FUNCTION "fcStdReportBatchStart" : Bool   // FC510, SCL
TITLE = Standard batch report start
{ S7_Optimized_Access := 'FALSE' }
AUTHOR : Boris
VERSION : 2.0
// 10/01/08 BC - Function needs to be called at batch start
//  Constant, used in all standard report FB and FC
   VAR_INPUT
      iInLineNo : Int;   // Line number
      iInMixerNo : Int;   // Mixer number
      sInFormulaName : String[254];   // Recipe name
      sInFormulaDescription : String[254];   // Recipe Description
      iInFormulaID : Int;   // Recipe ID
      iInBatchNumber : Int;   // Batch number
      sInTimeStart : String[254];   // Start timestamp
      rInMixerTempStart : Real;   // Mixer temperature AT batch start
   END_VAR
   VAR_IN_OUT
      MixerReportOperation : "udtStdReportOperV2";   // Current report operation with header and status
   END_VAR
   VAR_TEMP
      iTemp : Int;
      bResult : Bool;
   END_VAR
   VAR CONSTANT
      ciMaxQueue : Int := 200;   // Elements in the queue
      ciMaxUID : Int := 30000;
      ciReportDisable : Int;   // Not ready
      ciReportReady : Int := 10;   // Ready to save to database
      ciReportSavingToDataBase : Int := 20;   // Saving in progress
      ciReportFailed : Int := 30;   // Saving failed
      ciReportSaved : Int := 40;   // Saved
   END_VAR
BEGIN

       // Write batch header (with UID) to the mixer report operation header
       #MixerReportOperation.iBatchUID := "fcStdReportNewBatchUID"(); // Generate new global batch uid
       #MixerReportOperation.Header.iLineNo := #iInLineNo;
       #MixerReportOperation.Header.iMixerNo := #iInMixerNo;
       #MixerReportOperation.Header.iStatus := 220; // Set batch in progress status
       #iTemp := BLKMOV (DSTBLK => #MixerReportOperation.Header.sName, SRCBLK := #sInFormulaName);
       #iTemp := BLKMOV (DSTBLK => #MixerReportOperation.Header.sDescription, SRCBLK := #sInFormulaDescription);    
       #MixerReportOperation.Header.iRecipeID := #iInFormulaID;
       #MixerReportOperation.Header.iBatchNumber := #iInBatchNumber;
       #iTemp := BLKMOV (DSTBLK => #MixerReportOperation.Header.sTimeStart, SRCBLK := #sInTimeStart);        
       #MixerReportOperation.Header.rMixerTemp := #rInMixerTempStart;

       // Clear command structure
       #MixerReportOperation.Command.iStep := 0;
       #MixerReportOperation.Command.iStatus := 0;
       #MixerReportOperation.Command.sName := "sEmpty";
       #MixerReportOperation.Command.iCode := 0;
       #MixerReportOperation.Command.iIngredientType := 0;
       #MixerReportOperation.Command.sTimeStart := "sEmpty";
       #MixerReportOperation.Command.sTimeFinish := "sEmpty";
       #MixerReportOperation.Command.rSetpoint := 0.0;
       #MixerReportOperation.Command.rActual := 0.0;
       #MixerReportOperation.Command.rTemperature := 0.0;

       // Clear footer structure
       #MixerReportOperation.Footer.iStatus := 0;
       #MixerReportOperation.Footer.rMixerTemp := 0.0;
       #MixerReportOperation.Footer.sTimeFinish := "sEmpty";

       // Set reporting status to report ready
       #MixerReportOperation.iReportingStatus := #ciReportReady;

       // Generate new global index to write    
       #iTemp := "fcStdReportGetWriteIndex"();            
       // Check queue index already used, return false from function to indicate error
       IF ("dbStdReportQueueV2".Operations["dbStdReportQueueV2".iIndexWrite].iReportingStatus = #ciReportSaved) OR ("dbStdReportQueueV2".Operations["dbStdReportQueueV2".iIndexWrite].iReportingStatus = #ciReportDisable) THEN
           #bResult := true;
       ELSE
           #bResult := false;
       END_IF;

       // Write batch header to the queue
       #iTemp := BLKMOV (DSTBLK => "dbStdReportQueueV2".Operations["dbStdReportQueueV2".iIndexWrite], SRCBLK := #MixerReportOperation);

       // Return false if overwriting previous report in the queue
       #fcStdReportBatchStart := #bResult;                                
       ENO := true;
END_FUNCTION

FUNCTION "fcStdReportBatchComplete" : Bool   // FC511, SCL
TITLE = Standard batch report complete
{ S7_Optimized_Access := 'FALSE' }
AUTHOR : Boris
VERSION : 2.0
// 10/01/08 BC - Function needs to be called at batch complete
//  Constant, used in all standard report FB and FC
   VAR_INPUT
      iInLineNo : Int;   // Line number
      iInMixerNo : Int;   // Mixer number
      rInMixerTempFinish : Real;   // Mixer temperature
      sInTimeFinish : String[254];   // Complete timestamp
      iInBatchStatus : Int;   // Batch status (if not yet set)
   END_VAR
   VAR_IN_OUT
      MixerReportOperation : "udtStdReportOperV2";   // Current report operation with header and status
   END_VAR
   VAR_TEMP
      iTemp : Int;
      bResult : Bool;
   END_VAR
   VAR CONSTANT
      ciMaxQueue : Int := 200;   // Elements in the queue
      ciMaxUID : Int := 30000;
      ciReportDisable : Int;   // Not ready
      ciReportReady : Int := 10;   // Ready to save to database
      ciReportSavingToDataBase : Int := 20;   // Saving in progress
      ciReportFailed : Int := 30;   // Saving failed
      ciReportSaved : Int := 40;   // Saved
   END_VAR
BEGIN

       // Check batchUID, generate new if needed
       IF (#MixerReportOperation.iBatchUID = 0) THEN
           // Something went wrong - batch completed, but BatchUID is not set
           // Most likely it will be empty batch with only footer
           #MixerReportOperation.iBatchUID := "fcStdReportNewBatchUID"(); // Generate new global batch uid
           #MixerReportOperation.Header.iStatus := 220; // Set header to InProgress
       END_IF;

       // Clear command structure
       #MixerReportOperation.Command.iStep := 0;
       #MixerReportOperation.Command.iStatus := 0;
       #MixerReportOperation.Command.sName := "sEmpty";
       #MixerReportOperation.Command.iCode := 0;
       #MixerReportOperation.Command.iIngredientType := 0;
       #MixerReportOperation.Command.sTimeStart := "sEmpty";
       #MixerReportOperation.Command.sTimeFinish := "sEmpty";
       #MixerReportOperation.Command.rSetpoint := 0.0;
       #MixerReportOperation.Command.rActual := 0.0;
       #MixerReportOperation.Command.rTemperature := 0.0;

       // Write foter structure to the mixer operation report strucuture
       // If status not set yet - set it. Keep old status if it was previously set
       IF (#MixerReportOperation.Footer.iStatus = 0) THEN
           #MixerReportOperation.Footer.iStatus := #iInBatchStatus;
       END_IF;
       #MixerReportOperation.Footer.rMixerTemp := #rInMixerTempFinish;
       #iTemp := BLKMOV (DSTBLK => #MixerReportOperation.Footer.sTimeFinish, SRCBLK := #sInTimeFinish);                             
       #MixerReportOperation.Header.iLineNo := #iInLineNo;
       #MixerReportOperation.Header.iMixerNo := #iInMixerNo;

       // Set reporting status to report ready
       #MixerReportOperation.iReportingStatus := #ciReportReady;

       // Generate new global index to write    
       #iTemp := "fcStdReportGetWriteIndex"();  
       // Check queue index already used, return false from function to indicate error
       IF ("dbStdReportQueueV2".Operations["dbStdReportQueueV2".iIndexWrite].iReportingStatus = #ciReportSaved) OR ("dbStdReportQueueV2".Operations["dbStdReportQueueV2".iIndexWrite].iReportingStatus = #ciReportDisable) THEN
           #bResult := true;
       ELSE
           #bResult := false;
       END_IF;

       // Write batch header to the queue
       #iTemp := BLKMOV (DSTBLK => "dbStdReportQueueV2".Operations["dbStdReportQueueV2".iIndexWrite], SRCBLK := #MixerReportOperation);

       // Clear mixer operation report header strucutre
       #MixerReportOperation.iBatchUID := 0;
       #MixerReportOperation.Header.iLineNo := #iInLineNo;
       #MixerReportOperation.Header.iMixerNo := #iInMixerNo;
       #MixerReportOperation.Header.sName := "sEmpty";
       #MixerReportOperation.Header.sDescription := "sEmpty";
       #MixerReportOperation.Header.iRecipeID := 0;
       #MixerReportOperation.Header.iBatchNumber := 0;
       #MixerReportOperation.Header.iStatus := 0;
       #MixerReportOperation.Header.sTimeStart := "sEmpty";
       #MixerReportOperation.Header.rMixerTemp := 0.0;

       // Clear footer structure
       #MixerReportOperation.Footer.iStatus := 0;
       #MixerReportOperation.Footer.rMixerTemp := 0.0;
       #MixerReportOperation.Footer.sTimeFinish := "sEmpty";

       #MixerReportOperation.iReportingStatus := 0;

       // Return false if overwriting previous report in the queue
       #fcStdReportBatchComplete := #bResult;                                  
       ENO := true;
END_FUNCTION

FUNCTION "fcStdReportOper" : Bool   // FC512, SCL
TITLE = Standard batch report store operation
{ S7_Optimized_Access := 'FALSE' }
AUTHOR : Boris
VERSION : 2.0
// 10/01/08 BC - Function needs to be called at batch complete
//  Constant, used in all standard report FB and FC
   VAR_INPUT
      iInLineNo : Int;   // Line number
      iInMixerNo : Int;   // Mixer number
      iInStepNumber : Int;   // Command step number (0 if outside the recipe)
      iInCommandStatus : Int;   // Command delivery status
      sInCommandName : String[254];   // Command/Ingredient string name
      iInCommandCode : Int;   // Comand/Ingredient code
      iInCommandIngredientType : Int;   // Igredient type code
      sInCommandTimeStart : String[254];   // Delivery start time string
      sInCommandTimeFinish : String[254];   // Delivery comlete time string
      rInCommandSetpoint : Real;   // Delivery set point
      rInCommandActual : Real;   // Delivered actual
      rInCommandTemperature : Real;   // Ingredient temperature
   END_VAR
   VAR_IN_OUT
      MixerReportOperation : "udtStdReportOperV2";   // Current report operation with header and status
   END_VAR
   VAR_TEMP
      iTemp : Int;
      bResult : Bool;
   END_VAR
   VAR CONSTANT
      ciMaxQueue : Int := 200;   // Elements in the queue
      ciMaxUID : Int := 30000;
      ciReportDisable : Int;   // Not ready
      ciReportReady : Int := 10;   // Ready to save to database
      ciReportSavingToDataBase : Int := 20;   // Saving in progress
      ciReportFailed : Int := 30;   // Saving failed
      ciReportSaved : Int := 40;   // Saved
   END_VAR
BEGIN

       // Check batchUID, generate new if needed
       IF (#MixerReportOperation.iBatchUID = 0) THEN
           // Looks like we running test ingredient recipe
           #MixerReportOperation.Header.iStatus := 200; // Set header to TestRecipe
       END_IF;

       // Not normal situation - header status not set, assume test ingredient
       IF (#MixerReportOperation.Header.iStatus = 0) THEN
           #MixerReportOperation.Header.iStatus := 200; // Set header to TestRecipe
       END_IF;

       // Check if we running test recipe, idicated by header status
       IF (#MixerReportOperation.Header.iStatus = 200) THEN
           // Check if it's not intermediate weight        
           IF (#MixerReportOperation.Command.iStatus <> 1000) THEN    
               #iTemp := "fcStdReportNewBatchUID"(); // Generate new global batch uid
           END_IF;

           // Clear mixer operation report header structure
           #MixerReportOperation.Header.sName := "sEmpty";
           #MixerReportOperation.Header.sDescription := "sEmpty";
           #MixerReportOperation.Header.iRecipeID := 0;
           #MixerReportOperation.Header.iBatchNumber := 0;
           #MixerReportOperation.Header.sTimeStart := "sEmpty";
           #MixerReportOperation.Header.rMixerTemp := 0.0;

           // Clear footer structure        
           #MixerReportOperation.Footer.iStatus := 0;
           #MixerReportOperation.Footer.rMixerTemp := 0.0;
           #MixerReportOperation.Footer.sTimeFinish := "sEmpty";
       END_IF;

       // Set batch header 
       #MixerReportOperation.Header.iLineNo := #iInLineNo;
       #MixerReportOperation.Header.iMixerNo := #iInMixerNo;

       // Write command structure to the Mixer report operation structure
       #MixerReportOperation.Command.iStep := #iInStepNumber;
       #MixerReportOperation.Command.iStatus := #iInCommandStatus;
       #iTemp := BLKMOV (DSTBLK => #MixerReportOperation.Command.sName, SRCBLK := #sInCommandName);
       #MixerReportOperation.Command.iCode := #iInCommandCode;
       #MixerReportOperation.Command.iIngredientType := #iInCommandIngredientType;
       #iTemp := BLKMOV (DSTBLK => #MixerReportOperation.Command.sTimeStart, SRCBLK := #sInCommandTimeStart);
       #iTemp := BLKMOV (DSTBLK => #MixerReportOperation.Command.sTimeFinish, SRCBLK := #sInCommandTimeFinish);
       #MixerReportOperation.Command.rSetpoint := #rInCommandSetpoint;
       #MixerReportOperation.Command.rActual := #rInCommandActual;
       #MixerReportOperation.Command.rTemperature := #rInCommandTemperature;                                

       // Set reporting status to report ready
       #MixerReportOperation.iReportingStatus := #ciReportReady;

       // Generate new global index to write    
       #iTemp := "fcStdReportGetWriteIndex"();    
       // Check queue index already used, return false from function to indicate error
       IF ("dbStdReportQueueV2".Operations["dbStdReportQueueV2".iIndexWrite].iReportingStatus = #ciReportSaved) OR ("dbStdReportQueueV2".Operations["dbStdReportQueueV2".iIndexWrite].iReportingStatus = #ciReportDisable) THEN
           #bResult := true;
       ELSE
           #bResult := false;
       END_IF;

       // Write batch header to the queue
       #iTemp := BLKMOV (DSTBLK => "dbStdReportQueueV2".Operations["dbStdReportQueueV2".iIndexWrite], SRCBLK := #MixerReportOperation);

       // Return false if overwriting previous report in the queue
       #fcStdReportOper := #bResult;                 
       ENO := true;
END_FUNCTION

FUNCTION "fcStdReportBatchStatus" : Void   // FC513, SCL
TITLE = Standard batch report set batch status
{ S7_Optimized_Access := 'FALSE' }
AUTHOR : Boris
VERSION : 2.0
// Constant, used in all standard report FB and FC
   VAR_INPUT
      iInLineNo : Int;   // Line number
      iInMixerNo : Int;   // Mixer number
      iInBatchStatus : Int;   // Batch status to set
   END_VAR
   VAR_IN_OUT
      MixerReportOperation : "udtStdReportOperV2";   // Current report operation with header and status
   END_VAR
   VAR_TEMP
      iTemp : Int;
      bResult : Bool;
   END_VAR
   VAR CONSTANT
      ciMaxQueue : Int := 200;   // Elements in the queue
      ciMaxUID : Int := 30000;
      ciReportDisable : Int;   // Not ready
      ciReportReady : Int := 10;   // Ready to save to database
      ciReportSavingToDataBase : Int := 20;   // Saving in progress
      ciReportFailed : Int := 30;   // Saving failed
      ciReportSaved : Int := 40;   // Saved
   END_VAR
BEGIN

       // Write batch header
       #MixerReportOperation.Header.iLineNo := #iInLineNo;
       #MixerReportOperation.Header.iMixerNo := #iInMixerNo;

       // If status not set yet - set it. Keep old status if it was previously set
       IF (#MixerReportOperation.Footer.iStatus = 0) THEN
           #MixerReportOperation.Footer.iStatus := #iInBatchStatus;
       END_IF;

       ENO := true;
END_FUNCTION

FUNCTION "fcStdReportNewBatchUID" : Int   // FC514, SCL
TITLE = Standard batch report generates and return new batchUID
{ S7_Optimized_Access := 'FALSE' }
AUTHOR : Boris
VERSION : 2.0
// Constant, used in all standard report FB and FC
   VAR_TEMP
      i : Int;
   END_VAR
   VAR CONSTANT
      ciMaxQueue : Int := 200;   // Elements in the queue
      ciMaxUID : Int := 30000;
      ciReportDisable : Int;   // Not ready
      ciReportReady : Int := 10;   // Ready to save to database
      ciReportSavingToDataBase : Int := 20;   // Saving in progress
      ciReportFailed : Int := 30;   // Saving failed
      ciReportSaved : Int := 40;   // Saved
   END_VAR
BEGIN

       // Generate new global batch uid
       #i := "dbStdReportQueueV2".iGlobalBatchUID + 1;
       IF (#i > #ciMaxUID) THEN
          #i := 1;
       END_IF;  
       "dbStdReportQueueV2".iGlobalBatchUID := #i;

       #fcStdReportNewBatchUID := "dbStdReportQueueV2".iGlobalBatchUID;
       ENO := true;
END_FUNCTION

FUNCTION "fcStdReportGetWriteIndex" : Int   // FC515, SCL
TITLE = Standard batch report get queue write index
{ S7_Optimized_Access := 'FALSE' }
AUTHOR : Boris
VERSION : 2.0
// Constant, used in all standard report FB and FC
   VAR_TEMP
      i : Int;
   END_VAR
   VAR CONSTANT
      ciMaxQueue : Int := 200;   // Elements in the queue
      ciMaxUID : Int := 30000;
      ciReportDisable : Int;   // Not ready
      ciReportReady : Int := 10;   // Ready to save to database
      ciReportSavingToDataBase : Int := 20;   // Saving in progress
      ciReportFailed : Int := 30;   // Saving failed
      ciReportSaved : Int := 40;   // Saved
   END_VAR
BEGIN

       // Generate new global index to write    
       #i := "dbStdReportQueueV2".iIndexWrite + 1;      
       // Check queue index at the end of the queue
       IF (#i > #ciMaxQueue) THEN
           #i := 1;
       END_IF;               
       "dbStdReportQueueV2".iIndexWrite := #i;           

       #fcStdReportGetWriteIndex := "dbStdReportQueueV2".iIndexWrite;
       ENO := true;
END_FUNCTION

// folder: Resources/Process

FUNCTION_BLOCK "fbRetentiveTimer"   // FB385, LAD
TITLE = Retentive Timer Block
{ S7_Optimized_Access := 'TRUE' }
AUTHOR : DMC
FAMILY : LowLevel
VERSION : 0.1
// //  This is a retentive count-up timer.
// //  IN makes it count.  It does not reset when IN is off.
// //  RESET resets the time to 0.  
// //  bInPT is the time setpoint.
// //  bOutEnabled is true when the time has the setpoint
// //  bOutET is the elapsed time.
   VAR_INPUT
      IN : Bool;   // Counter Starts when this is true
      RESET : Bool;   // Counter Resets when this is true
      PT : Time;   // Time setpoint
   END_VAR
   VAR_OUTPUT
      Q : Bool;   // True when Elapsed time > Time Setpoint
      ET : Time;   // Elapsed Time
   END_VAR
   VAR
      "Timer" : IEC_TIMER;   // Timer
      tInternalTime : Time;   // Internal Time
      tTimer1ET : Time;   // Elapsed Time of Timer 1
      ET_DINT : DInt;   // Elapsed Time as a double integer
      bTON_Timer : Bool;
   END_VAR
   VAR_TEMP
      diTemp1 : DInt;   // Temp Double int
      diTemp2 : DInt;   // Temp Double int
      diTemp3 : DInt;   // Temp Double int
      tTemp : Time;
   END_VAR
   VAR CONSTANT
      ctMaxTime : Time := T#24D_20H_31M_23S_647MS;   // Max possible time
   END_VAR
BEGIN

REGION Network 1: Keep resetting internal time while not counting
   // IF (NOT IN) THEN
   //     tInternalTime := tInternalTime + Timer1.ET;
   // END_IF;
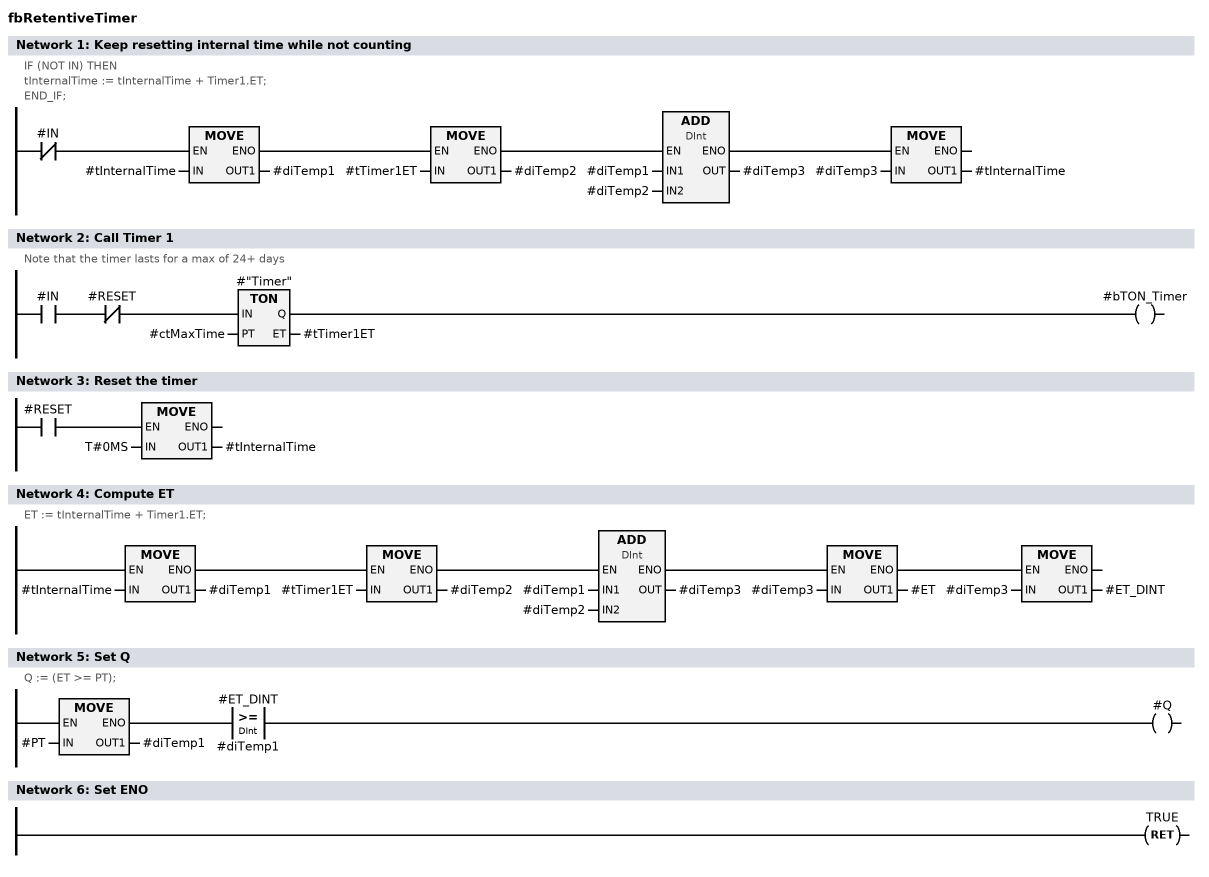
   RUNG wire#powerrail
      I_Contact( #IN )
      { S7_GenerateENO := "TRUE" } Move(in := #tInternalTime, out1 => #diTemp1)
      { S7_GenerateENO := "TRUE" } Move(in := #tTimer1ET, out1 => #diTemp2)
      { S7_Templates := "SrcType := DInt"; S7_GenerateENO := "TRUE" } Add(in1 := #diTemp1, in2 := #diTemp2, out => #diTemp3)
      { S7_GenerateENO := "TRUE" } Move(in := #diTemp3, out1 => #tInternalTime)
   END_RUNG
   // the same network as SCL:
   // ENO of a box is taken as its EN; it also drops when the box reports an error
   IF NOT #IN THEN
       #diTemp1 := #tInternalTime;
       #diTemp2 := #tTimer1ET;
       #diTemp3 := #diTemp1 + #diTemp2;
       #tInternalTime := #diTemp3;
   END_IF;
END_REGION

REGION Network 2: Call Timer 1
   // Note that the timer lasts for a max of 24+ days
   #"Timer".TON(IN := #IN AND NOT #RESET, PT := #ctMaxTime, ET => #tTimer1ET);
   #bTON_Timer := #"Timer".Q;
END_REGION

REGION Network 3: Reset the timer
   RUNG wire#powerrail
      Contact( #RESET )
      { S7_GenerateENO := "TRUE" } Move(in := T#0MS, out1 => #tInternalTime)
   END_RUNG
   // the same network as SCL:
   IF #RESET THEN #tInternalTime := T#0MS; END_IF;
END_REGION

REGION Network 4: Compute ET
   // ET := tInternalTime + Timer1.ET;
   RUNG wire#powerrail
      { S7_GenerateENO := "TRUE" } Move(in := #tInternalTime, out1 => #diTemp1)
      { S7_GenerateENO := "TRUE" } Move(in := #tTimer1ET, out1 => #diTemp2)
      { S7_Templates := "SrcType := DInt"; S7_GenerateENO := "TRUE" } Add(in1 := #diTemp1, in2 := #diTemp2, out => #diTemp3)
      { S7_GenerateENO := "TRUE" } Move(in := #diTemp3, out1 => #ET)
      { S7_GenerateENO := "TRUE" } Move(in := #diTemp3, out1 => #ET_DINT)
   END_RUNG
   // the same network as SCL:
   // ENO of a box is taken as its EN; it also drops when the box reports an error
   #diTemp1 := #tInternalTime;
   #diTemp2 := #tTimer1ET;
   #diTemp3 := #diTemp1 + #diTemp2;
   #ET := #diTemp3;
   #ET_DINT := #diTemp3;
END_REGION

REGION Network 5: Set Q
   // Q := (ET >= PT);
   RUNG wire#powerrail
      { S7_GenerateENO := "TRUE" } Move(in := #PT, out1 => #diTemp1)
      { S7_Templates := "SrcType := DInt" } GE_Contact(in1 := #ET_DINT, in2 := #diTemp1)
      Coil( #Q )
   END_RUNG
   // the same network as SCL:
   // ENO of a box is taken as its EN; it also drops when the box reports an error
   #diTemp1 := #PT;
   #Q := #ET_DINT >= #diTemp1;
END_REGION

REGION Network 6: Set ENO
   RUNG wire#powerrail
      ReturnCoil( TRUE )
   END_RUNG
   // the same network as SCL:
   ENO := TRUE;
   RETURN;
END_REGION
END_FUNCTION_BLOCK

// ===== library: MasterCopy "Copy of BUFFER_SEARCH" =====

FUNCTION_BLOCK "BUFFER_SEARCH"   // FB229, SCL
TITLE = BUFFER_SEARCH
{ S7_Optimized_Access := 'FALSE' }
AUTHOR : hugo
FAMILY : BUFFER
NAME : BSEARCH
VERSION : 1.4
// this function will search for a string STR in an array of byte starting at position pos.
//   the function needs to be called: buffer_search(adr("array"),sizeof("array"), STR, POS, IGN);
//   because this function works with pointers its very time efficient and it needs no extra memory.
//   The function returns the position of the first character of the string in the array if found.
//   a -1 is returned if the string is not found in the array.
//   when IGN = TRUE, STR must be in capital letters and the search is case insensitv.
//   
// VERSION : '1.4'
// AUTHOR  : hugo
// NAME    : BSEARCH
// FAMILY  : BUFFER
   VAR_INPUT
      PT : Variant;
      _pt AT PT : Struct
         DBNr : Word;
         Adr : DWord;
      END_STRUCT;
      SIZE : Int;
      STR : String[254];
      _str AT STR : Struct
         length : Byte;
         act_length : Byte;
         str : Array[1..254] of Byte;
      END_STRUCT;
      POS : Int;
      IGN : Bool;
   END_VAR
   VAR_OUTPUT
      _SEARCH : Int;
   END_VAR
   VAR_TEMP
      ps : Int;   // POINTER TO ARRAY[0..255] OF BYTE;
      chx : Byte;
      i : Int;
      end : Int;
      k : Int;
      lx : Int;
      tPT : Int;
      c : Char;
      searchByte : Byte;
   END_VAR
BEGIN


   #tPT := DWORD_TO_INT(SHR(IN:=SHL(IN:=#_pt.Adr,N:=8),N:=11));

   #ps := 1;    //ADR(str);
   #lx := BYTE_TO_INT(#_str.act_length);  //LEN(str);
   #end := MIN(IN1:=#SIZE - #lx, IN2:= #SIZE - 1);
   #lx := #lx - 1;
   FOR #i := #POS TO #end DO
     FOR #k := 0 TO #lx DO
       //IF (_str.str[ps+k] <> ign) AND (_str.str[ps+k] <> WORD_TO_BLOCK_DB(_pt.DBNr).DB[tPT+i+k]) THEN EXIT; END_IF;
       IF #IGN THEN 
         #chx := TO_UPPER(WORD_TO_BLOCK_DB(#_pt.DBNr).#tPT+#i+#k)); 
         #searchByte:= TO_UPPER(#_str.str[#ps+#k]);
         #c:=BYTE_TO_CHAR(#searchByte);  
       ELSE 
         #chx := WORD_TO_BLOCK_DB(#_pt.DBNr).#tPT+#i+#k); 
         #searchByte:= #_str.str[#ps+#k];
         #c:=BYTE_TO_CHAR(#searchByte);
       END_IF;

       IF #searchByte <> #chx THEN 
         EXIT; 
       END_IF;
     END_FOR;
     IF #k > #lx THEN
       #_SEARCH := #i;
       RETURN;
     END_IF;
   END_FOR;
   #_SEARCH := -1;


   (* revision History

   hm 5. mar. 2008 rev 1.0
     original version

   hm  16. mar. 2008 rev 1.1
     chaged type of input size to uint

   hm  13. may. 2008 rev 1.2
     changed type of pointer to array[1..32767]
     changed size of string to STRING_LENGTH

   hm  12. nov. 2009 rev 1.3
     limit end to array size

   hm  25. jan. 2011 rev 1.4
     ign = True will now ignore case
     return -1 if nothing found

   TMJ  4. May. 2013 rev 1.5
     function wasn't working at all. fixed comparison logic
   *)
END_FUNCTION_BLOCK

(* ===== HMI "HMI_RT_1" =====

HMI tags "Default tag table"
   "val1" : Int, internal
   "val2" : Int, internal
   "val3" : Int, internal

ScreenModuleEditorView "Faceplate_1" 640x480
   IOField "I/O field_1" at 10,10 size 133x28; FormatPattern 9
      ProcessValue <- "myBool"
*)